TYPE ST_TcMatSimObjectDataAreaInfo_2 :
STRUCT
	pPlcVar: PVOID;
	pModuleProcImg: PVOID;
	nSize: UDINT;
	nDataAreaId: UDINT;
	eDataAreaType: E_TcMatSimDataAreaType;
END_STRUCT
END_TYPE

(* stored: Version 1.1.0.1, ProductVersion 3.1.4020.12
   DUT ST_TcMatSimObjectDataAreaInfo_2: Id {bc77eeab-8b99-4a23-9f80-720fda817ef7} *)
